// TIA Portal V21 export
DATA_BLOCK "ComunicazioneS7_St1_Robopack"   // DB9001
{ S7_Optimized_Access := 'FALSE' }
   VAR
      Send : Struct
         Digitali : Array[0..31] of Bool;
         "DInt" : Array[0..19] of DInt;
         "Real" : Array[0..19] of Real;
      END_STRUCT;
      Receive : Struct
         Digitali : Array[0..31] of Bool;
         "DInt" : Array[0..19] of DInt;
         "Real" : Array[0..19] of Real;
      END_STRUCT;
   END_VAR
BEGIN
   Send.Digitali[0] := FALSE;   // Watchdog
   Send.Digitali[1..31] := FALSE;
   Send."DInt"[0] := 0;   // Watchdog
   Send."DInt"[1..19] := 0;
   Send."Real"[0..19] := 0.0;
   Receive.Digitali[0] := FALSE;   // Watchdog
   Receive.Digitali[1..31] := FALSE;
   Receive."DInt"[0] := 0;   // Watchdog
   Receive."DInt"[1..19] := 0;
   Receive."Real"[0..19] := 0.0;
END_DATA_BLOCK
